// TwinCAT 3 PLC project Carro_Basico_PLC
// ProgramVersion: 3.1.4024.0
// libraries:
//   Tc2_Standard, * (Beckhoff Automation GmbH)
//   Tc2_System, * (Beckhoff Automation GmbH)
//   Tc3_Module, * (Beckhoff Automation GmbH)
//   VisuDialogs, * (System)
// project tree:
//   / GlobalTextList.TcGTLO (not stored), PlcTask.TcTTO (not stored), Visualization Manager.TcVMO (not stored)
//   POUs/ FB_Blink.TcPOU, FB_Carro_DRC_LD.TcPOU, FB_Carro_GRF_LD.TcPOU, FB_Carro_GRF_SFC.TcPOU, FB_Carro_GRF_ST.TcPOU (not stored), MAIN.TcPOU
//   VISUs/ V_Carro.TcVIS

// ---- POUs/FB_Blink.TcPOU
// Square wave oscillator
FUNCTION_BLOCK FB_Blink
VAR_INPUT
    Enable: BOOL := TRUE; // Enables oscillator
    TimeOn: TIME := T#500MS; // Duration of HIGH phase
    TimeOff: TIME := T#500MS; // Duration of LOW phase
END_VAR
VAR_OUTPUT
    Q: BOOL; // Oscillating output
END_VAR
VAR
    Timer: TON;
    ToggleEdge: R_TRIG;
    PhaseDuration: TIME;
END_VAR

// Guard Clause: deterministic reset
IF NOT Enable THEN
    Q := FALSE;
    Timer(IN := FALSE);
    ToggleEdge(CLK := FALSE);
    RETURN;
END_IF;

// Select current phase duration
IF Q THEN
    PhaseDuration := TimeOn;
ELSE
    PhaseDuration := TimeOff;
END_IF;

// Execute Timer
Timer(
    IN := TRUE, 
    PT := PhaseDuration
);

// Toggle logic on timer completion
ToggleEdge(CLK := Timer.Q);

// State toggle on each timer completion
IF ToggleEdge.Q THEN
    Q := NOT Q;
    // Reset timer to restart on next scan
    Timer(IN := FALSE);
END_IF;

END_FUNCTION_BLOCK

// ---- POUs/FB_Carro_DRC_LD.TcPOU
FUNCTION_BLOCK FB_Carro_DRC_LD
// Transcripción «indirecta» del diagrama de relés y contactos (DRC -> LD)
VAR_INPUT
    ManiobrasTotales: UINT := 2;
    TiempoEspera: TIME := T#2S;
END_VAR
VAR_OUTPUT
    ManiobrasPendientes: UINT;
    TiempoPendiente: TIME;
END_VAR
VAR
    // Estasdos actuales
    EnIzquierda: BOOL;
    
    // Estados futuros
    MarchaDerechaFuturo: BOOL;
    MarchaIzquierdaFuturo: BOOL;
    
    // Bloques funcionales
    FlancoPulsadorMarcha: R_TRIG;
    Intermitencia: FB_Blink;
    TemporizadorEspera: TON;
    ContadorManiobras: CTD := (Q := TRUE);
    
    // Entradas
    i_PulsadorMarcha AT %I*: BOOL;
    i_FinalCarreraIzquierda AT %I*: BOOL := TRUE;
    i_FinalCarreraDerecha AT %I*: BOOL;
    
    // Salidas
    o_MarchaIzquierda AT %I*: BOOL;
    o_MarchaDerecha AT %I*: BOOL;
    o_LamparaMarcha AT %I*: BOOL;
END_VAR

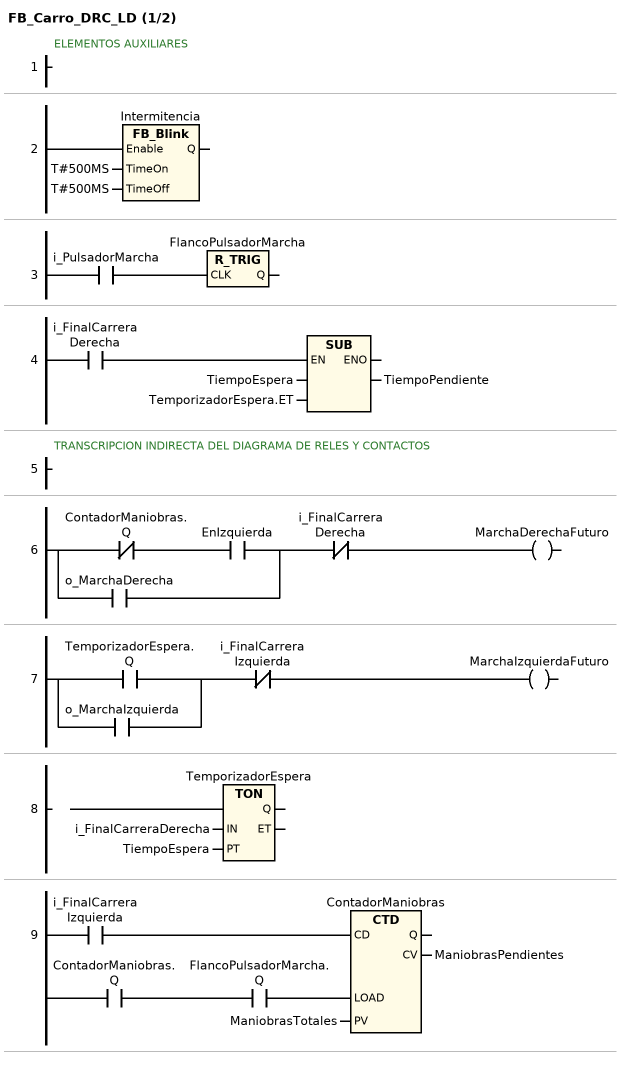
// NETWORK 1
// ELEMENTOS AUXILIARES

// NETWORK 2
Intermitencia(Enable := TRUE, TimeOn := T#500MS, TimeOff := T#500MS); // FB_Blink

// NETWORK 3
FlancoPulsadorMarcha(CLK := i_PulsadorMarcha); // R_TRIG

// NETWORK 4
IF i_FinalCarreraDerecha THEN TiempoPendiente := TiempoEspera - TemporizadorEspera.ET; END_IF

// NETWORK 5
// TRANSCRIPCION INDIRECTA DEL DIAGRAMA DE RELES Y CONTACTOS

// NETWORK 6
MarchaDerechaFuturo := (NOT ContadorManiobras.Q AND EnIzquierda OR o_MarchaDerecha) AND NOT i_FinalCarreraDerecha;

// NETWORK 7
MarchaIzquierdaFuturo := (TemporizadorEspera.Q OR o_MarchaIzquierda) AND NOT i_FinalCarreraIzquierda;

// NETWORK 8
TemporizadorEspera(IN := i_FinalCarreraDerecha, PT := TiempoEspera); // TON

// NETWORK 9
ContadorManiobras(
    CD := i_FinalCarreraIzquierda,
    LOAD := ContadorManiobras.Q AND FlancoPulsadorMarcha.Q,
    PV := ManiobrasTotales,
    CV => ManiobrasPendientes); // CTD

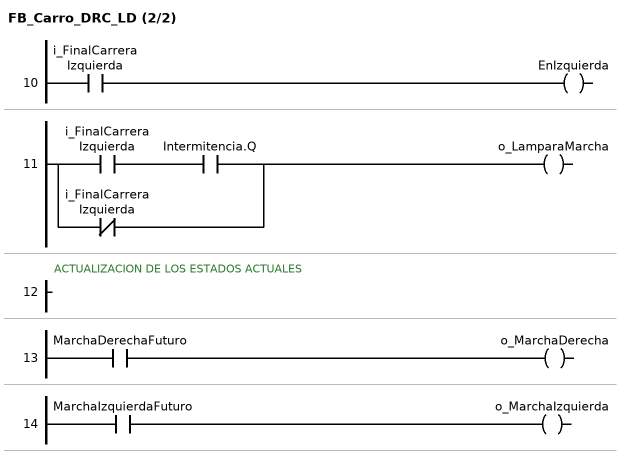
// NETWORK 10
EnIzquierda := i_FinalCarreraIzquierda;

// NETWORK 11
o_LamparaMarcha := i_FinalCarreraIzquierda AND Intermitencia.Q OR NOT i_FinalCarreraIzquierda;

// NETWORK 12
// ACTUALIZACION DE LOS ESTADOS ACTUALES

// NETWORK 13
o_MarchaDerecha := MarchaDerechaFuturo;

// NETWORK 14
o_MarchaIzquierda := MarchaIzquierdaFuturo;

END_FUNCTION_BLOCK

// ---- POUs/FB_Carro_GRF_LD.TcPOU
FUNCTION_BLOCK FB_Carro_GRF_LD
// Transcripción del grafcet (GRF -> LD) [Usando células eléctricas de memoria]
VAR_INPUT
    ManiobrasTotales: UINT := 2;
    TiempoEspera: TIME := T#2S;
END_VAR
VAR_OUTPUT
    ManiobrasPendientes: UINT;
    TiempoPendiente: TIME;
END_VAR
VAR
    TiempoActual: TIME;
    
    // Variables propias del GRF
    S0x: BOOL := TRUE; // Etapa inicial
    S1x, S2x, S3x, S4x: BOOL; // Etapas no-iniciales
    t0, t1, t2, t3, t4, t4a: BOOL; // Transiciones
    S2t, S2_t: TIME; // S2.t y S2._t
    
    // Bloques funcionales
    FlancoPulsadorMarcha: R_TRIG;
    Intermitencia: FB_Blink;
    
    // Entradas
    i_PulsadorMarcha AT %I*: BOOL;
    i_FinalCarreraIzquierda AT %I*: BOOL := TRUE;
    i_FinalCarreraDerecha AT %I*: BOOL;
    
    // Salidas
    o_MarchaIzquierda AT %I*: BOOL;
    o_MarchaDerecha AT %I*: BOOL;
    o_LamparaMarcha AT %I*: BOOL;
END_VAR

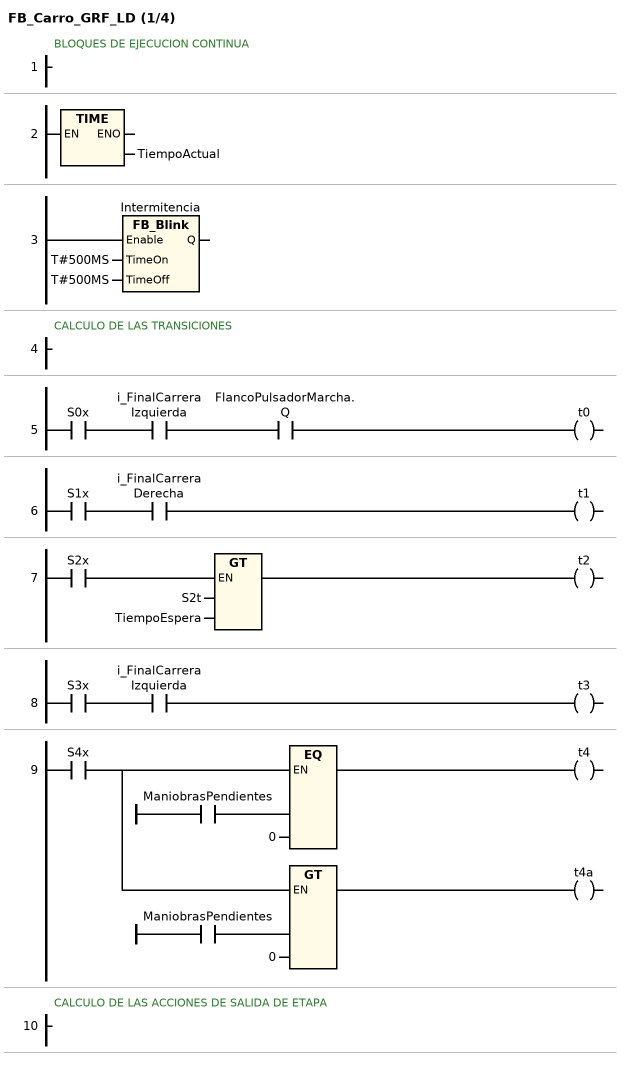
// NETWORK 1
// BLOQUES DE EJECUCION CONTINUA

// NETWORK 2
TiempoActual := TIME();

// NETWORK 3
Intermitencia(Enable := TRUE, TimeOn := T#500MS, TimeOff := T#500MS); // FB_Blink

// NETWORK 4
// CALCULO DE LAS TRANSICIONES

// NETWORK 5
t0 := S0x AND i_FinalCarreraIzquierda AND FlancoPulsadorMarcha.Q;

// NETWORK 6
t1 := S1x AND i_FinalCarreraDerecha;

// NETWORK 7
t2 := S2x AND S2t > TiempoEspera;

// NETWORK 8
t3 := S3x AND i_FinalCarreraIzquierda;

// NETWORK 9
t4 := S4x AND ManiobrasPendientes = 0;
t4a := S4x AND ManiobrasPendientes > 0;

// NETWORK 10
// CALCULO DE LAS ACCIONES DE SALIDA DE ETAPA

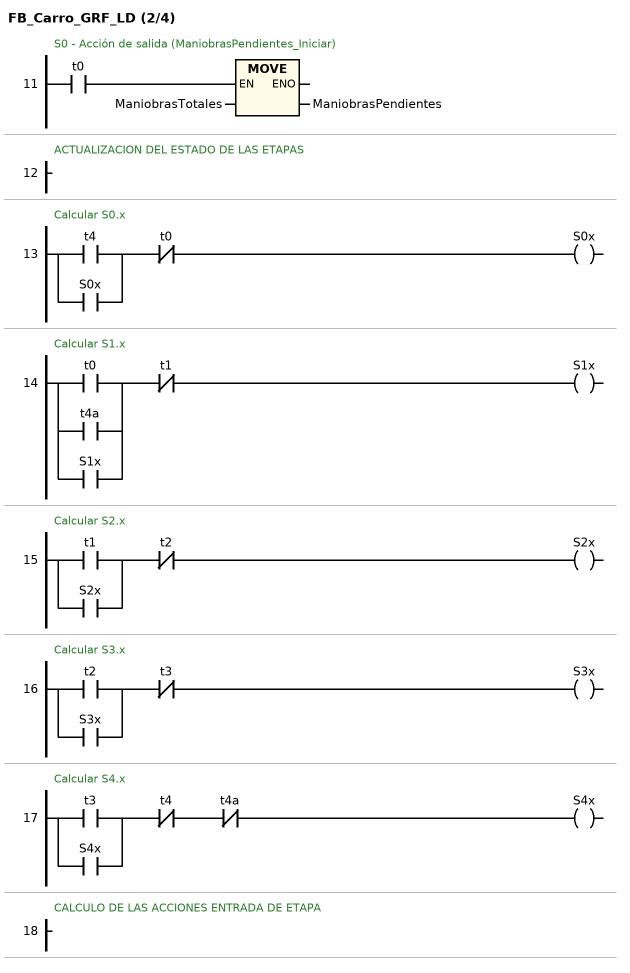
// NETWORK 11
// S0 - Acción de salida (ManiobrasPendientes_Iniciar)
IF t0 THEN ManiobrasPendientes := ManiobrasTotales; END_IF

// NETWORK 12
// ACTUALIZACION DEL ESTADO DE LAS ETAPAS

// NETWORK 13
// Calcular S0.x
S0x := (t4 OR S0x) AND NOT t0;

// NETWORK 14
// Calcular S1.x
S1x := (t0 OR t4a OR S1x) AND NOT t1;

// NETWORK 15
// Calcular S2.x
S2x := (t1 OR S2x) AND NOT t2;

// NETWORK 16
// Calcular S3.x
S3x := (t2 OR S3x) AND NOT t3;

// NETWORK 17
// Calcular S4.x
S4x := (t3 OR S4x) AND NOT t4 AND NOT t4a;

// NETWORK 18
// CALCULO DE LAS ACCIONES ENTRADA DE ETAPA

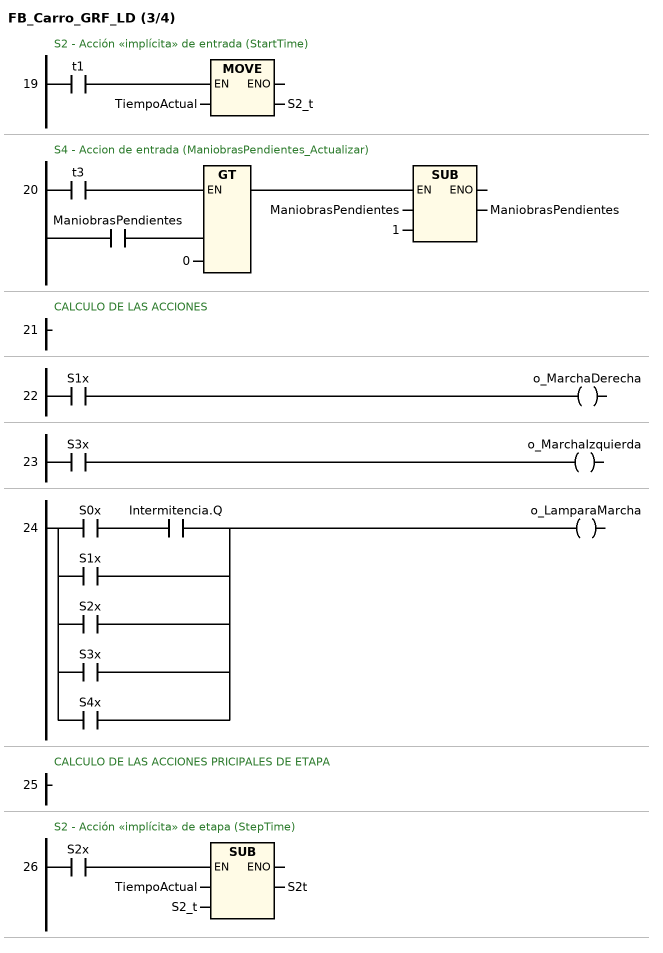
// NETWORK 19
// S2 - Acción «implícita» de entrada (StartTime)
IF t1 THEN S2_t := TiempoActual; END_IF

// NETWORK 20
// S4 - Accion de entrada (ManiobrasPendientes_Actualizar)
IF t3 AND ManiobrasPendientes > 0 THEN ManiobrasPendientes := ManiobrasPendientes - 1; END_IF

// NETWORK 21
// CALCULO DE LAS ACCIONES

// NETWORK 22
o_MarchaDerecha := S1x;

// NETWORK 23
o_MarchaIzquierda := S3x;

// NETWORK 24
o_LamparaMarcha := S0x AND Intermitencia.Q OR S1x OR S2x OR S3x OR S4x;

// NETWORK 25
// CALCULO DE LAS ACCIONES PRICIPALES DE ETAPA

// NETWORK 26
// S2 - Acción «implícita» de etapa (StepTime)
IF S2x THEN S2t := TiempoActual - S2_t; END_IF

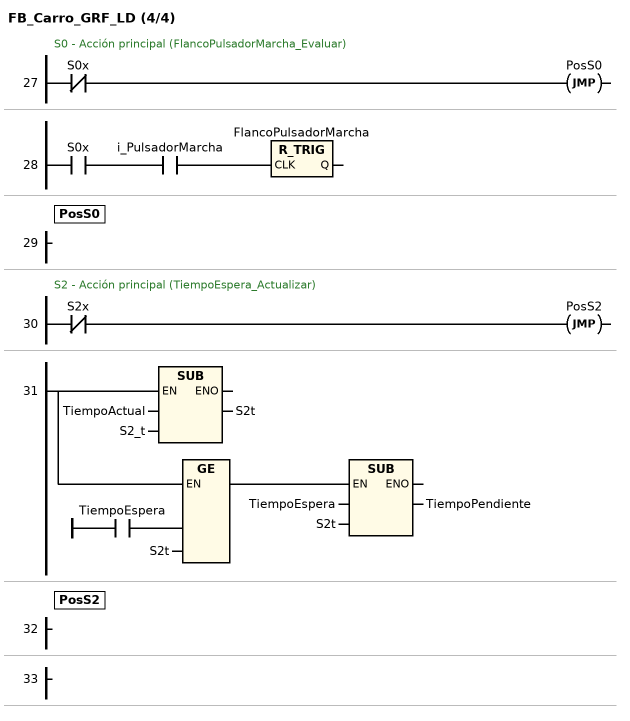
// NETWORK 27
// S0 - Acción principal (FlancoPulsadorMarcha_Evaluar)
IF NOT S0x THEN JMP PosS0; END_IF

// NETWORK 28
FlancoPulsadorMarcha(CLK := S0x AND i_PulsadorMarcha); // R_TRIG

// NETWORK 29
PosS0: ;

// NETWORK 30
// S2 - Acción principal (TiempoEspera_Actualizar)
IF NOT S2x THEN JMP PosS2; END_IF

// NETWORK 31
S2t := TiempoActual - S2_t;
IF TiempoEspera >= S2t THEN TiempoPendiente := TiempoEspera - S2t; END_IF

// NETWORK 32
PosS2: ;

// NETWORK 33

END_FUNCTION_BLOCK

// ---- POUs/FB_Carro_GRF_SFC.TcPOU
FUNCTION_BLOCK FB_Carro_GRF_SFC
// Transcripción del grafcet (GRF -> SFC)
VAR_INPUT
    ManiobrasTotales: UINT := 2;
    TiempoEspera: TIME := T#2S;
END_VAR
VAR_OUTPUT
    ManiobrasPendientes: UINT;
    TiempoPendiente: TIME;
END_VAR
VAR
    // Bloques funcionales
    FlancoPulsadorMarcha: R_TRIG;
    Intermitencia: FB_Blink;
    
    // Entradas
    i_PulsadorMarcha AT %I*: BOOL;
    i_FinalCarreraIzquierda AT %I*: BOOL := TRUE;
    i_FinalCarreraDerecha AT %I*: BOOL;
    
    // Salidas
    o_MarchaIzquierda AT %I*: BOOL;
    o_MarchaDerecha AT %I*: BOOL;
    o_LamparaMarcha AT %I*: BOOL;
END_VAR

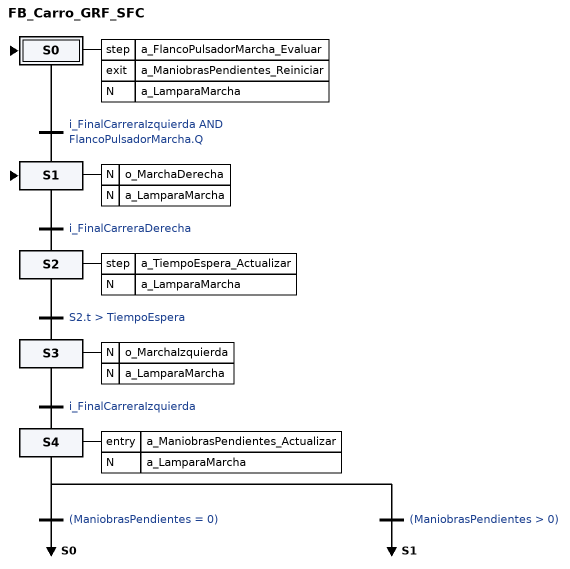
INITIAL_STEP S0:
    a_FlancoPulsadorMarcha_Evaluar(N);  // step action
    a_ManiobrasPendientes_Reiniciar(P0);  // exit action
    a_LamparaMarcha(N);
END_STEP
TRANSITION FROM S0 TO S1
    := i_FinalCarreraIzquierda AND FlancoPulsadorMarcha.Q;
END_TRANSITION
STEP S1:
    o_MarchaDerecha(N);
    a_LamparaMarcha(N);
END_STEP
TRANSITION FROM S1 TO S2
    := i_FinalCarreraDerecha;
END_TRANSITION
STEP S2:
    a_TiempoEspera_Actualizar(N);  // step action
    a_LamparaMarcha(N);
END_STEP
TRANSITION FROM S2 TO S3
    := S2.t > TiempoEspera;
END_TRANSITION
STEP S3:
    o_MarchaIzquierda(N);
    a_LamparaMarcha(N);
END_STEP
TRANSITION FROM S3 TO S4
    := i_FinalCarreraIzquierda;
END_TRANSITION
STEP S4:
    a_ManiobrasPendientes_Actualizar(P1);  // entry action
    a_LamparaMarcha(N);
END_STEP
TRANSITION FROM S4 TO S0
    := (ManiobrasPendientes = 0);
END_TRANSITION
TRANSITION FROM S4 TO S1
    := (ManiobrasPendientes > 0);
END_TRANSITION

ACTION a_FlancoPulsadorMarcha_Evaluar:
FlancoPulsadorMarcha(CLK := i_PulsadorMarcha);
END_ACTION

ACTION a_LamparaMarcha:
Intermitencia(Enable := S0.x);

o_LamparaMarcha := (S0.x AND Intermitencia.Q) OR S1.x OR S2.x OR S3.x OR S4.x;
END_ACTION

ACTION a_ManiobrasPendientes_Actualizar:
IF (ManiobrasPendientes > 0) THEN
    ManiobrasPendientes := ManiobrasPendientes - 1;
END_IF;
END_ACTION

ACTION a_ManiobrasPendientes_Reiniciar:
ManiobrasPendientes := ManiobrasTotales;
END_ACTION

ACTION a_TiempoEspera_Actualizar:
IF TiempoEspera >= S2.t THEN
    TiempoPendiente := TiempoEspera - S2.t;
END_IF;
END_ACTION

END_FUNCTION_BLOCK

// ---- POUs/MAIN.TcPOU
PROGRAM MAIN
VAR
    // Carro: FB_Carro_DRC_LD;
    Carro: FB_Carro_GRF_SFC;
    // Carro: FB_Carro_GRF_ST;
    // Carro: FB_Carro_GRF_LD;
END_VAR

Carro();

END_PROGRAM

// ---- VISUs/V_Carro.TcVIS
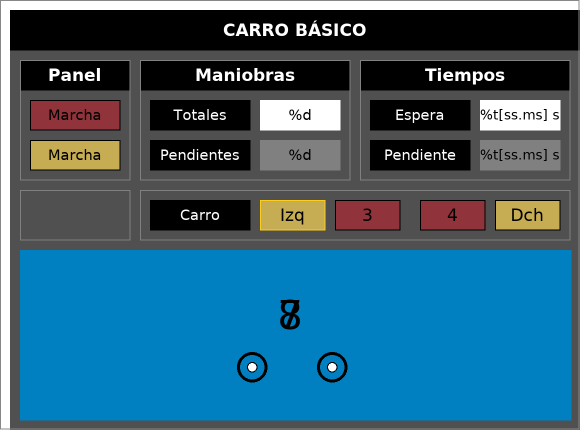
VISUALIZATION V_Carro  // 580x430
    Rectangle (10,50 570x380)
    Rectangle (140,190 430x50)
    Rectangle (20,60 110x30), "Panel"
    Rectangle (20,60 110x120)
    Rectangle (360,60 210x30), "Tiempos"
    Rectangle (360,60 210x120)
    Rectangle (10,10 570x40), "CARRO BÁSICO"
    RoundedRectangle (370,100 100x30), "Espera"
    Rectangle (140,60 210x30), "Maniobras"
    Rectangle (480,100 80x30), "%t[ss.ms] s", text variable: MAIN.Carro.TiempoEspera
        OnMouseClick: write the text variable via Default
    RoundedRectangle (370,140 100x30), "Pendiente"
    Rectangle (480,140 80x30), "%t[ss.ms] s", text variable: MAIN.Carro.TiempoPendiente
        OnMouseClick: write the text variable via Default
    Rectangle (30,100 90x30), "Marcha", colour toggle: MAIN.Carro.o_LamparaMarcha
        tap MAIN.Carro.o_LamparaMarcha
    Rectangle (30,140 90x30), "Marcha", colour toggle: MAIN.Carro.i_PulsadorMarcha
        toggle MAIN.Carro.i_PulsadorMarcha
    Rectangle (140,60 210x120)
    RoundedRectangle (150,100 100x30), "Totales"
    Rectangle (260,100 80x30), "%d", text variable: MAIN.Carro.ManiobrasTotales
        OnMouseClick: write the text variable via Default
    RoundedRectangle (150,140 100x30), "Pendientes"
    Rectangle (260,140 80x30), "%d", text variable: MAIN.Carro.ManiobrasPendientes
        OnMouseClick: write the text variable via Default
    Rectangle (20,250 551x170)
    Polyline (477,390)
    Polygon (105,385), colour toggle: MAIN.Carro.i_FinalCarreraIzquierda
        p2738717112: SEL (MAIN.Carro.i_FinalCarreraIzquierda, 0, 5)
        toggle MAIN.Carro.i_FinalCarreraIzquierda
    Polygon (435,385), colour toggle: MAIN.Carro.i_FinalCarreraDerecha
        p2738717112: SEL (MAIN.Carro.i_FinalCarreraDerecha, 0, 5)
        toggle MAIN.Carro.i_FinalCarreraDerecha
    Group (211,281 158x98), invisible if: MAIN.Carro.i_FinalCarreraIzquierda AND MAIN.Carro.i_FinalCarreraDerecha
        p3560616238: SEL (MAIN.Carro.i_FinalCarreraDerecha, SEL (MAIN.Carro.i_FinalCarreraIzquierda, 0, -125), 125)
        Polygon (0,0)
        Polygon (115,80)
        Group (106,71 28x28)
            Ellipse (0,0 30x30)
            Ellipse (10,10 10x10)
        Polygon (35,80)
        Group (26,71 28x28)
            Ellipse (0,0 30x30)
            Ellipse (10,10 10x10)
    Rectangle (270,295 40x40), "8", tooltip "Marcha derecha", invisible if: NOT MAIN.Carro.o_MarchaDerecha
        p3560616238: SEL (MAIN.Carro.i_FinalCarreraDerecha, SEL (MAIN.Carro.i_FinalCarreraIzquierda, 0, -125), 125)
    Rectangle (270,295 40x40), "7", invisible if: NOT MAIN.Carro.o_MarchaIzquierda
        p3560616238: SEL (MAIN.Carro.i_FinalCarreraDerecha, SEL (MAIN.Carro.i_FinalCarreraIzquierda, 0, -125), 125)
    RoundedRectangle (150,200 100x30), "Carro"
    Rectangle (335,200 65x30), "3", colour toggle: MAIN.Carro.o_MarchaIzquierda
        toggle MAIN.Carro.o_MarchaIzquierda
    Rectangle (420,200 65x30), "4", colour toggle: MAIN.Carro.o_MarchaDerecha
        toggle MAIN.Carro.o_MarchaDerecha
    Rectangle (260,200 65x30), "Izq", colour toggle: MAIN.Carro.i_FinalCarreraIzquierda
        toggle MAIN.Carro.i_FinalCarreraIzquierda
    Rectangle (495,200 65x30), "Dch", colour toggle: MAIN.Carro.i_FinalCarreraDerecha
        toggle MAIN.Carro.i_FinalCarreraDerecha
    Rectangle (20,190 110x50)
END_VISUALIZATION
